PROGRAM MAIN
VAR
	m : INT;
END_VAR

m := m + 1;
PrgMqttCom();

END_PROGRAM

(* stored: Version 1.1.0.1, ProductVersion 3.1.4021.12
   POU MAIN: Id {d85bfd96-1b0c-45d0-a980-65fe0d2ef94f}, SpecialFunc None *)
